FUNCTION_BLOCK FB_Siemens_SendDp_Test EXTENDS TcUnit.FB_TestSuite

Test_ProcessDataControl();
Test_ProcessDataStatus();

METHOD Test_ProcessDataControl : REFERENCE TO FB_Test
VAR
	fbDevice 						: FB_Siemens_SendDp;
	
	nExpectdRcvData					: WORD;
	nExpectdRcvSequenceNumber		: WORD;
	nExpectdRcvCrc					: WORD;	
	
	nActualRcvData					: WORD;
	nActualRcvSequenceNumber		: WORD;
	nActualRcvCrc					: WORD;
		
	stExpectedControlData 			: ST_Siemens_SendDp_Control;		
	stActualControlData				: ST_Siemens_SendDp_Control;	
	nDigitalOutputs: INT;
END_VAR
TEST('Process data to control structure');

//Arrange
nExpectdRcvData := 16#A1B2;					
nExpectdRcvSequenceNumber := 16#C3D4;		
nExpectdRcvCrc := 16#E5F6;		
	
F_Memcpy(ADR(stExpectedControlData), ADR(nExpectdRcvData), 2, FALSE);
F_Memcpy(ADR(stExpectedControlData) + 2, ADR(nExpectdRcvSequenceNumber), 2, FALSE);
F_Memcpy(ADR(stExpectedControlData) + 4, ADR(nExpectdRcvCrc), 2, FALSE);

fbDevice.pControl := ADR(stExpectedControlData);

//Act
fbDevice.GetControlData();

stActualControlData := fbDevice.stControl;

//Assert
			 
AssertEquals(Expected := nExpectdRcvData,
             Actual := stActualControlData.nRcvData,
             Message := 'RcvData is not correct');
			 
AssertEquals(Expected := nExpectdRcvSequenceNumber,
             Actual := stActualControlData.nRcvSequenceNumber,
             Message := 'SequenceNumber is not correct');
			 
AssertEquals(Expected := nExpectdRcvCrc,
             Actual := stActualControlData.nRcvCrc,
             Message := 'RcvCrc is not correct');			 
			 
TEST_FINISHED();


TEST('Process data to control structure SWAP');

//Arrange
nExpectdRcvData := 16#A1B2;					
nExpectdRcvSequenceNumber := 16#C3D4;		
nExpectdRcvCrc := 16#E5F6;		
	
F_Memcpy(ADR(stExpectedControlData), ADR(nExpectdRcvData), 2, TRUE);
F_Memcpy(ADR(stExpectedControlData) + 2, ADR(nExpectdRcvSequenceNumber), 2, TRUE);
F_Memcpy(ADR(stExpectedControlData) + 4, ADR(nExpectdRcvCrc), 2, TRUE);

fbDevice.pControl := ADR(stExpectedControlData);

fbDevice.stConfig.bSwapProcessData := TRUE;

//Act
fbDevice.GetControlData();

stActualControlData := fbDevice.stControl;

//Assert
			 
AssertEquals(Expected := nExpectdRcvData,
             Actual := stActualControlData.nRcvData,
             Message := 'RcvData is not correct');
			 
AssertEquals(Expected := nExpectdRcvSequenceNumber,
             Actual := stActualControlData.nRcvSequenceNumber,
             Message := 'SequenceNumber is not correct');
			 
AssertEquals(Expected := nExpectdRcvCrc,
             Actual := stActualControlData.nRcvCrc,
             Message := 'RcvCrc is not correct');				 
			 
TEST_FINISHED();
END_METHOD

METHOD Test_ProcessDataStatus : REFERENCE TO FB_Test
VAR
	fbDevice 						: FB_Siemens_SendDp;
	
	nExpectedBoolData				: WORD;
	nExpectedSendInt00				: INT;
	nExpectedSendInt01				: INT;
	nExpectedSendData				: WORD;
	nExpectedSendSequenceNumber		: WORD;	
	nExpectedSendCrc				: WORD;
	
	stExpectedStatusData 			: ST_Siemens_SendDp_Status;		
	stActualStatusData 				: ST_Siemens_SendDp_Status;	
END_VAR
TEST('Assign status structure to process data');

//Arrange
nExpectedBoolData := 16#A1B2;	
nExpectedSendInt00 := UINT_TO_INT(16#C3D4);
nExpectedSendInt01 := UINT_TO_INT(16#E5F6);	
nExpectedSendData := 16#B6A5;					
nExpectedSendSequenceNumber := 16#D4C3;	
nExpectedSendCrc := 16#E2F1;		

F_Memcpy(ADR(fbDevice.stStatus), ADR(nExpectedBoolData), 2, FALSE);
F_Memcpy(ADR(fbDevice.stStatus) + 2, ADR(nExpectedSendInt00), 2, FALSE);
F_Memcpy(ADR(fbDevice.stStatus) + 4, ADR(nExpectedSendInt01), 2, FALSE);
F_Memcpy(ADR(fbDevice.stStatus) + 6, ADR(nExpectedSendData), 2, FALSE);
F_Memcpy(ADR(fbDevice.stStatus) + 8, ADR(nExpectedSendSequenceNumber), 2, FALSE);
F_Memcpy(ADR(fbDevice.stStatus) + 10, ADR(nExpectedSendCrc), 2, FALSE);

fbDevice.pStatus := ADR(stActualStatusData);

//Act
fbDevice.SetStatusData();

//Assert
AssertEquals(Expected := nExpectedBoolData,
             Actual := stActualStatusData.nSendBoolData,
             Message := 'SendBoolData is not correct');
	 
AssertEquals(Expected := nExpectedSendInt00,
             Actual := stActualStatusData.nSendInt00,
             Message := 'SendInt00 is not correct');	

AssertEquals(Expected := nExpectedSendInt01,
             Actual := stActualStatusData.nSendInt01,
             Message := 'SendInt01 is not correct');
			 
AssertEquals(Expected := nExpectedSendData,
             Actual := stActualStatusData.nSendData,
             Message := 'SendData is not correct');
	 
AssertEquals(Expected := nExpectedSendSequenceNumber,
             Actual := stActualStatusData.nSendSequenceNumber,
             Message := 'SendSequenceNumber is not correct');	

AssertEquals(Expected := nExpectedSendCrc,
             Actual := stActualStatusData.nSendCrc,
             Message := 'SendCrc is not correct');
					 			 
TEST_FINISHED();


TEST('Assign status structure to process data SWAP');

//Arrange
nExpectedBoolData := 16#A1B2;	
nExpectedSendInt00 := UINT_TO_INT(16#C3D4);
nExpectedSendInt01 := UINT_TO_INT(16#E5F6);	
nExpectedSendData := 16#B6A5;					
nExpectedSendSequenceNumber := 16#D4C3;	
nExpectedSendCrc := 16#E2F1;		

F_Memcpy(ADR(fbDevice.stStatus), ADR(nExpectedBoolData), 2, TRUE);
F_Memcpy(ADR(fbDevice.stStatus) + 2, ADR(nExpectedSendInt00), 2, TRUE);
F_Memcpy(ADR(fbDevice.stStatus) + 4, ADR(nExpectedSendInt01), 2, TRUE);
F_Memcpy(ADR(fbDevice.stStatus) + 6, ADR(nExpectedSendData), 2, TRUE);
F_Memcpy(ADR(fbDevice.stStatus) + 8, ADR(nExpectedSendSequenceNumber), 2, TRUE);
F_Memcpy(ADR(fbDevice.stStatus) + 10, ADR(nExpectedSendCrc), 2, TRUE);

fbDevice.pStatus := ADR(stActualStatusData);

fbDevice.stConfig.bSwapProcessData := TRUE;

//Act
fbDevice.SetStatusData();

//Assert
AssertEquals(Expected := nExpectedBoolData,
             Actual := stActualStatusData.nSendBoolData,
             Message := 'SendBoolData is not correct');
	 
AssertEquals(Expected := nExpectedSendInt00,
             Actual := stActualStatusData.nSendInt00,
             Message := 'SendInt00 is not correct');	

AssertEquals(Expected := nExpectedSendInt01,
             Actual := stActualStatusData.nSendInt01,
             Message := 'SendInt01 is not correct');
			 
AssertEquals(Expected := nExpectedSendData,
             Actual := stActualStatusData.nSendData,
             Message := 'SendData is not correct');
	 
AssertEquals(Expected := nExpectedSendSequenceNumber,
             Actual := stActualStatusData.nSendSequenceNumber,
             Message := 'SendSequenceNumber is not correct');	

AssertEquals(Expected := nExpectedSendCrc,
             Actual := stActualStatusData.nSendCrc,
             Message := 'SendCrc is not correct');
					 			 
TEST_FINISHED();
END_METHOD

END_FUNCTION_BLOCK

(* stored: Version 1.1.0.1, ProductVersion 3.1.4024.12
   POU FB_Siemens_SendDp_Test: Id {4cb7908e-4774-0fba-29a0-4e26524aaea5}, SpecialFunc None
   Method Test_ProcessDataControl: Id {9333f770-922f-0b09-0409-d08e8a30371d}
   Method Test_ProcessDataStatus: Id {1e943c56-2fdc-0916-0f21-3fa952259a67} *)
